// TIA Portal V20 export
TYPE "typeSequenceControlNodeJobInterface"
// stored: Namespace Unit1.Em3
   STRUCT
      commands : "Unit1.Em3.typeSequenceControlNodeJobInterfaceCommands";
      monitoring { S7_SetPoint := 'True'} : "Unit1.Em3.typeSequenceControlNodeJobInterfaceMonitoring";
   END_STRUCT;
END_TYPE
